PROGRAM main
VAR
	Enable AT %QX0.0 : bool;
	DelayTimer : TON;
	Output AT %QX0.1 : bool;
	DelayTimer_ET : time;
	DelayTimer_ElapsedSeconds AT %MD0 : dint;
END_VAR

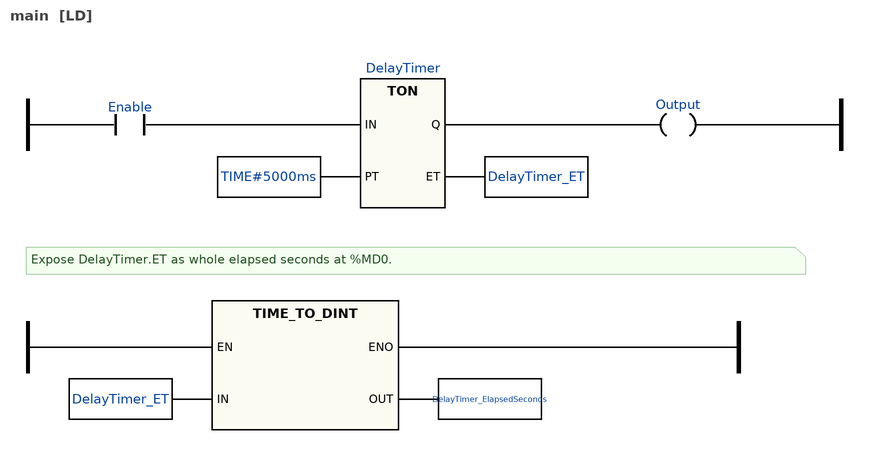
(* LD diagram, written out as Structured Text *)
DelayTimer(IN := Enable, PT := TIME#5000ms);
DelayTimer_ET := DelayTimer.ET;
Output := DelayTimer.Q;
(* Expose DelayTimer.ET as whole elapsed seconds at %MD0. *)
DelayTimer_ElapsedSeconds := TIME_TO_DINT(DelayTimer_ET);
END_PROGRAM
